//{attribute 'qualified_only'}
VAR_GLOBAL
	{attribute 'pytmc' := '
    pv: LXLHN:VAC:OVERRIDE
	field: ZNAM OVERRIDE OFF ;
	field: ONAM OVERRIDE ON ;
	'}
	xSystemOverrideMode_LAS : BOOL := FALSE;
END_VAR

(* stored: Version 1.1.0.1, ProductVersion 3.1.4022.18
   GVL GVL_BTS_OVERRIDES: Id {f55be108-cc20-45ff-a5e5-29ed15a33c84} *)
